{attribute 'qualified_only'}
{attribute 'strict'}
TYPE E_ScannerResult :
(
	None := 0,
	GoodRead := 1,
	NoRead := 2,
	LabelConflict := 3,
	NoData := 4,
	Overflow := 5 
);
END_TYPE

(* stored: Version 1.1.0.1, ProductVersion 3.1.4022.10
   DUT E_ScannerResult: Id {edca643a-e3d2-4dc7-aa86-7fc4882ab256} *)
